(* IEC 61131-3 sources: verifaps-lib/geteta/examples/rttcounter, 2 files *)

(* ---- OneCnt.st ---- *)
PROGRAM OneCnt
VAR s : INT; END_VAR

VAR_OUTPUT
    c : INT;
END_VAR

    s := s + 1;
    c :=  s;

END_PROGRAM

(* ---- TwoCnt.st ---- *)
PROGRAM TwoCnt
VAR_OUTPUT
    c : INT;
END_VAR

    c := c + 2;

END_PROGRAM
